VISUALIZATION Visu_Liftkabine  // 1024x768
END_VISUALIZATION

(* stored: Version 1.1.0.1
   Visu Visu_Liftkabine: Id {a9491971-ba43-4b2b-a709-8f22390ed508} *)
